// TIA Portal V17 export
// export: Created 2025-03-05T08:02:02.1697367Z, ExportSetting WithDefaults, DisplayName Totally Integrated Automation Portal, DisplayVersion V17 Update 8, DisplayName TIA Portal Openness, DisplayVersion V17 Update 8, DisplayName TIA Portal Version Control Interface, DisplayVersion V17, DisplayName SINAMICS Startdrive Advanced, DisplayVersion V17 SP2, DisplayName SINAMICS Startdrive G110M, G120, G120C, G120D, G120P, G115D, DisplayVersion V17 SP2, DisplayName SINAMICS Startdrive G130, G150, S120, S150, SINAMICS MV, S210, DisplayVersion V17 SP2, DisplayName STEP 7 Professional, DisplayVersion V17 Update 8, DisplayName SINUMERIK ONE STEP 7 Toolbox, DisplayVersion V17 Update 12, DisplayName SINUMERIK 840D sl STEP 7 Toolbox, DisplayVersion V17 Update 12, DisplayName STEP 7 Safety, DisplayVersion V17 Update 6, DisplayName WinCC Advanced, DisplayVersion V17 Update 8
TYPE "LBP_typeMcp483StandardOutput"
TITLE = MCP 483 image / Imagen de MCP 483 / MCP 483 Abbild
// Output image of MCP 483 / Imagen de salida de MCP 483 / Ausgangsabbild von MCP 483
// stored: IsFailsafeCompliant false
   STRUCT
      auto : Bool;
      mda : Bool;
      teachIn : Bool;
      jog : Bool;
      inc1 : Bool;
      inc10 : Bool;
      inc100 : Bool;
      inc1000 : Bool;
      inc10000 : Bool;
      incVar : Bool;
      refPoint : Bool;
      repos : Bool;
      cycleStop : Bool;
      cycleStart : Bool;
      feedrateStop : Bool;
      feedrateStart : Bool;
      spindleStop : Bool;
      spindleStart : Bool;
      singleBlock : Bool;
      axis10 : Bool;   // R10
      axis7 : Bool;   // R7
      axis4 : Bool;   // R4
      axisX : Bool;   // R1
      minus : Bool;   // R13
      plus : Bool;   // R15
      axis6 : Bool;   // R6
      axis8 : Bool;   // R8
      axis9 : Bool;   // R9
      axis11 : Bool;   // R11
      mcsWcs : Bool;   // R12
      axis5 : Bool;   // R5
      axisZ : Bool;   // R3
      axisY : Bool;   // R2
      customerKey15 : Bool;   // T15
      customerKey14 : Bool;   // T14
      customerKey13 : Bool;   // T13
      customerKey12 : Bool;   // T12
      customerKey11 : Bool;   // T11
      customerKey10 : Bool;   // T10
      customerKey9 : Bool;   // T9
      customerKey8 : Bool;   // T8
      customerKey7 : Bool;   // T7
      customerKey6 : Bool;   // T6
      customerKey5 : Bool;   // T5
      customerKey4 : Bool;   // T4
      customerKey3 : Bool;   // T3
      customerKey2 : Bool;   // T2
      customerKey1 : Bool;   // T1
      rapidTraverse : Bool;   // R14
      reset : Bool;
      reserved62 : Bool;
      reserved63 : Bool;
      reserved64 : Bool;
      reserved65 : Bool;
      reserved66 : Bool;
      reserved67 : Bool;
      optionalKey1 : Bool;   // KT-OUT1, reserviert / KT-OUT1, reserved / KT-OUT1, reservado
      optionalKey2 : Bool;   // KT-OUT2, reserviert / KT-OUT2, reserved / KT-OUT2, reservado
      optionalKey3 : Bool;   // KT-OUT3, reserviert / KT-OUT3, reserved / KT-OUT3, reservado
      optionalKey4 : Bool;   // KT-OUT4, reserviert / KT-OUT4, reserved / KT-OUT4, reservado
      optionalKey5 : Bool;   // KT-OUT5, reserviert / KT-OUT5, reserved / KT-OUT5, reservado
      optionalKey6 : Bool;   // KT-OUT6, reserviert / KT-OUT6, reserved / KT-OUT6, reservado
      reserved76 : Bool;
      reserved77 : Bool;
   END_STRUCT;
END_TYPE
